# EPICS autosave request: iocBoot/ioc13raman/auto_settings.req
file "ccd_settings.req",                P=13Raman:, C=ccd1
file "scan_settings.req",               P=13Raman:, S=scan1
file "scan_settings.req",               P=13Raman:, S=scan2
file "scan_settings.req",               P=13Raman:, S=scan3
file "scan_settings.req",               P=13Raman:, S=scan4
file "CARS_motor_settings.req",         P=13Raman:, M=m1
file "CARS_motor_settings.req",         P=13Raman:, M=m2
file "CARS_motor_settings.req",         P=13Raman:, M=m3
